// TwinCAT 3 PLC project SPT_Base_Types
// Title: SPT Base Types
// Company: Beckhoff Automation LLC
// ProjectVersion: 4.0.0.2
// Description: 4.0.0.2 I_InterfaceBase Generic base created 4.0.0.1 - removing other libs code
// libraries:
//   SPT Event Logger, * (Beckhoff Automation LLC)
//   Tc2_EtherCAT, * (Beckhoff Automation GmbH)
//   Tc2_Standard, * (Beckhoff Automation GmbH)
//   Tc2_System, * (Beckhoff Automation GmbH)
//   Tc2_Utilities, * (Beckhoff Automation GmbH)
//   Tc3_EventLogger, * (Beckhoff Automation GmbH)
//   Tc3_JsonXml, * (Beckhoff Automation GmbH)
//   Tc3_PackML_V2, * (Beckhoff Automation GmbH)
// project tree:
//   Enums/ E_AlarmResponse.TcTLEO
//   Framework Base/ FB_BaseFB.TcPOU, FB_CyclicFB.TcPOU
//   / GlobalTextList.TcGTLO, Parameters_Tracing.TcGVL
//   Interfaces/ I_BaseFB.TcIO, I_CyclicFB.TcIO, I_InterfaceBase.TcIO
//   Project Information/ F_GetCompany.TcPOU, F_GetTitle.TcPOU, F_GetVersion.TcPOU
//   Tracing/ FB_TraceLog.TcPOU, Tracing.TcGVL
//   Version/ Global_Version.TcGVL
// real-time tasks:
//   TASK Task 3: cycle T#10ms, priority 1, ADS port 350

// ---- Enums/E_AlarmResponse.TcTLEO
{attribute 'qualified_only'}
{attribute 'strict'}
{attribute 'to_string'}
TYPE E_AlarmResponse : (
		Abort_ImmediateError,
		Abort_Immediate,
		Stop_Immediate,
		Stop_Controlled,
		Hold_Immediate,
		Hold_Controlled,
		Suspend_Immediate,
		Suspend_Controlled,
		NoResponse
	);
END_TYPE

// ---- Parameters_Tracing.TcGVL
{attribute 'qualified_only'}
VAR_GLOBAL CONSTANT
	TRACING_ENABLED						: BOOL	:= TRUE;
	MAX_LOG_ENTRIES_PER_SCAN			: UDINT := 100;
	ALLOW_DUPLICATE_SEQUENTIAL_MESSAGES : BOOL	:= FALSE;
END_VAR

// ---- Tracing/Tracing.TcGVL
{attribute 'qualified_only'}
VAR_GLOBAL
	GlobalTraceLog : FB_TraceLog;
END_VAR

// ---- Version/Global_Version.TcGVL
{attribute 'TcGenerated'}
{attribute 'no-analysis'}
{attribute 'linkalways'}
// This function has been automatically generated from the project information.
VAR_GLOBAL CONSTANT
	{attribute 'const_non_replaced'}
	stLibVersion_SPT_Base_Types : ST_LibVersion := (iMajor := 4, iMinor := 0, iBuild := 0, iRevision := 2, nFlags := 0, sVersion := '4.0.0.2');
END_VAR

// ---- Interfaces/I_BaseFB.TcIO
INTERFACE I_BaseFB EXTENDS I_InterfaceBase

PROPERTY Busy : BOOL
GET
END_GET
END_PROPERTY

PROPERTY Error : BOOL
GET
END_GET
END_PROPERTY

PROPERTY ErrorID : UDINT;
GET
END_GET
END_PROPERTY

END_INTERFACE

// ---- Interfaces/I_CyclicFB.TcIO
INTERFACE I_CyclicFB EXTENDS I_BaseFB

METHOD CyclicLogic
VAR_INPUT
END_VAR
END_METHOD

PROPERTY InitComplete : BOOL
GET
END_GET
END_PROPERTY

END_INTERFACE

// ---- Interfaces/I_InterfaceBase.TcIO
INTERFACE I_InterfaceBase EXTENDS __SYSTEM.IQueryInterface

END_INTERFACE

// ---- Tracing/FB_TraceLog.TcPOU
FUNCTION_BLOCK FINAL FB_TraceLog
VAR
  Event : FB_TcMessage;
  JsonParser : FB_JsonDomParser;
  TimeFormatter : FB_FormatString;
  MessagesSentThisScan : UDINT;
  Previous_AddEntrySource : T_MaxString;
  Previous_AddEntryMessage : T_MaxString;
  Previous_AddEntryFlags : UDINT;
  Previous_AddEntryJsonSource : T_MaxString;
  Previous_AddEntryJsonMessage : T_MaxString;
  Previous_AddEntryJsonFlags : UDINT;
  Previous_AddEntryJson : T_MaxString;
END_VAR

METHOD PRIVATE AddContext
VAR_INPUT
  Source : T_MaxString;
  Flags : UDINT;
END_VAR

VAR
  CurrentDCTime : DCTIMESTRUCT;
  DCTime100Nsec : WORD;
END_VAR
//Collect DC timestamp info and properly format string
CurrentDCTime := DCTIME64_TO_DCTIMESTRUCT(F_GetActualDcTime64());
DCTime100Nsec := CurrentDCTime.wNanoseconds / 100;
TimeFormatter(
  sFormat := '%2.2d:%2.2d:%2.2d.%3.3d%3.3d%1.1d',
  arg1 := F_WORD(CurrentDCTime.wHour),
  arg2 := F_WORD(CurrentDCTime.wMinute),
  arg3 := F_WORD(CurrentDCTime.wSecond),
  arg4 := F_WORD(CurrentDCTime.wMilliseconds),
  arg5 := F_WORD(CurrentDCTime.wMicroseconds),
  arg6 := F_WORD(DCTime100Nsec)
);

Event.ipArguments.AddString(TimeFormatter.sOut); //DC Timestamp string
Event.ipArguments.AddString(Source); //POU calling the Trace() function -- this should come automatically
Event.ipArguments.AddString(TwinCAT_SystemInfoVarList._TaskInfo[GETCURTASKINDEXEX()].TaskName); //Task which called the POU last
Event.ipArguments.AddUDInt(TwinCAT_SystemInfoVarList._TaskInfo[GETCURTASKINDEXEX()].CycleCount); //Cycle count of above task
Event.ipArguments.AddUDInt(Flags); //General-use flags (application dependent)
END_METHOD

METHOD PUBLIC AddEntry
VAR_INPUT
  Source : T_MaxString;
  Message : T_MaxString;
  Flags : UDINT;
END_VAR
{analysis -62}
IF NOT TracingAllowed THEN
  {analysis -90}
  RETURN;
END_IF

IF NOT Parameters_Tracing.ALLOW_DUPLICATE_SEQUENTIAL_MESSAGES THEN
  IF (MEMCMP(ADR(Source), ADR(Previous_AddEntrySource), SIZEOF(T_MaxString)) = 0)
       AND (MEMCMP(ADR(Message), ADR(Previous_AddEntryMessage), SIZEOF(T_MaxString)) = 0)
       AND (Flags = Previous_AddEntryFlags) THEN
    //This message is identical to the last message sent--ignore
    RETURN;
  END_IF
END_IF

Event.ipArguments.Clear().AddString(Message);
AddContext(Source := Source, Flags := Flags);
Event.Send(0);
MessagesSentThisScan := MessagesSentThisScan + 1;
MEMCPY(ADR(Previous_AddEntrySource), ADR(Source), SIZEOF(T_MaxString));
MEMCPY(ADR(Previous_AddEntryMessage), ADR(Message), SIZEOF(T_MaxString));
Previous_AddEntryFlags := Flags;
END_METHOD

METHOD PUBLIC AddEntryWithJson
VAR_INPUT
  Source : T_MaxString;
  Message : T_MaxString;
  Flags : UDINT;
  Json : T_MaxString;
END_VAR

VAR
  Document : SJsonValue;
  JsonAttribute : T_MaxString;
  TaskName : T_MaxString;
  temp : udint;
END_VAR

VAR_INST
  LastScanCount : UDINT;
  MessagesSentThisScan : UDINT;
  MissedMessages : UDINT;
  Throttled : BOOL;
END_VAR

VAR
  ThrottledNotificationString : T_MaxString;
  CurrentDCTime : DCTIMESTRUCT;
  DCTime100Nsec : WORD;
  DCTimeString : T_MaxString;
END_VAR
{analysis -62}
IF NOT TracingAllowed THEN
  RETURN;
END_IF

IF NOT Parameters_Tracing.ALLOW_DUPLICATE_SEQUENTIAL_MESSAGES THEN
  IF (MEMCMP(ADR(Source), ADR(Previous_AddEntryJsonSource), SIZEOF(T_MaxString)) = 0)
       AND (MEMCMP(ADR(Message), ADR(Previous_AddEntryJsonMessage), SIZEOF(T_MaxString)) = 0)
       AND (Flags = Previous_AddEntryJsonFlags)
       AND (MEMCMP(ADR(Json), ADR(Previous_AddEntryJson), SIZEOF(T_MaxString)) = 0) THEN
    //This message is identical to the last message sent--ignore
    RETURN;
  END_IF
END_IF

Event.ipArguments.Clear().AddString(Message);
AddContext(Source := Source, Flags := Flags);
Document := JsonParser.NewDocument();
JsonParser.AddJsonMember(Document, 'ExtendedInfo', Json);
JsonAttribute := JsonParser.GetJson(Document);
Event.SetJsonAttribute(JsonAttribute);
Event.Send(0);
MessagesSentThisScan := MessagesSentThisScan + 1;
MEMCPY(ADR(Previous_AddEntryJsonSource), ADR(Source), SIZEOF(T_MaxString));
MEMCPY(ADR(Previous_AddEntryJsonMessage), ADR(Message), SIZEOF(T_MaxString));
Previous_AddEntryFlags := Flags;
MEMCPY(ADR(Previous_AddEntryJsonMessage), ADR(Json), SIZEOF(T_MaxString));
END_METHOD

METHOD FB_init : BOOL
VAR_INPUT
  bInitRetains : BOOL; // if TRUE, the retain variables are initialized (warm start / cold start)
  bInCopyCode : BOOL; // if TRUE, the instance afterwards gets moved into the copy code (online change)
END_VAR

VAR
  hr : HRESULT;
END_VAR
{analysis -15}
IF NOT Event.EqualsToEventEntryEx(TC_EVENTS.Tracing.TraceEvent) THEN
  Event.CreateEx(TC_EVENTS.Tracing.TraceEvent, 0);
END_IF
END_METHOD

PROPERTY PRIVATE TracingAllowed : BOOL
GET
VAR_INST
  LastScanCount : UDINT;
  MissedMessages : UDINT;
  Throttled : BOOL;
END_VAR

VAR
  ThrottledNotificationString : T_MaxString;
END_VAR
{analysis -62}
IF NOT Parameters_Tracing.TRACING_ENABLED THEN
  TracingAllowed := FALSE;
  RETURN;
END_IF

IF TwinCAT_SystemInfoVarList._TaskInfo[GETCURTASKINDEXEX()].CycleCount = LastScanCount THEN
  //Trying to send multiple messages in same scan
  IF Throttled THEN
    MissedMessages := MissedMessages + 1;
    RETURN;
  ELSIF MessagesSentThisScan >= Parameters_Tracing.MAX_LOG_ENTRIES_PER_SCAN AND NOT Throttled THEN
    //Need to throttle messsage queue
    Event.ipArguments.Clear().AddString('Too many messages sent in single scan; tracing throttled.');
    Event.Send(0);
    MissedMessages := MissedMessages + 1;
    Throttled := TRUE;
    TracingAllowed := FALSE;
    RETURN;
  ELSE
    TracingAllowed := TRUE;
  END_IF
ELSE
  IF Throttled THEN
    ThrottledNotificationString := CONCAT('Missed ', CONCAT(TO_STRING(MissedMessages), ' throttled messages previously.'));
    Event.ipArguments.Clear().AddString(ThrottledNotificationString);
    Event.Send(0);
    MissedMessages := 0;
  END_IF

  LastScanCount := TwinCAT_SystemInfoVarList._TaskInfo[GETCURTASKINDEXEX()].CycleCount;
  MessagesSentThisScan := 0;
  Throttled := FALSE;
  TracingAllowed := TRUE;
END_IF
END_GET
END_PROPERTY

END_FUNCTION_BLOCK

// ---- Framework Base/FB_BaseFB.TcPOU
{attribute 'reflection'}
FUNCTION_BLOCK ABSTRACT FB_BaseFB IMPLEMENTS I_BaseFB
VAR
  {attribute 'instance-path'}
  {attribute 'noinit'}
  InstancePath : STRING;
END_VAR

// I_BaseFB
VAR
  _Busy : BOOL := TRUE;
  _Error : BOOL;
  _ErrorID : UDINT;
END_VAR

// Derivatives of FB_BaseFB can have code in the function block body

PROPERTY Busy : BOOL
GET
Busy := _Busy;
END_GET
END_PROPERTY

PROPERTY Error : BOOL
GET
Error := _Error;
END_GET
END_PROPERTY

PROPERTY ErrorID : UDINT
GET
ErrorID := _ErrorID;
END_GET
END_PROPERTY

METHOD PUBLIC Marker
VAR_INPUT
  Message : T_MaxString;
END_VAR
Tracing.GlobalTraceLog.AddEntry(InstancePath, Message, 1);
END_METHOD

METHOD PUBLIC Trace
VAR_INPUT
  Message : T_MaxString;
END_VAR
Tracing.GlobalTraceLog.AddEntry(InstancePath, Message, 0);
END_METHOD

METHOD PUBLIC TraceWithJson
VAR_INPUT
  Message : T_MaxString;
  Json : T_MaxString;
END_VAR
Tracing.GlobalTraceLog.AddEntryWithJson(
  InstancePath,
  Message,
  0,
  Json
);
END_METHOD

END_FUNCTION_BLOCK

// ---- Framework Base/FB_CyclicFB.TcPOU
{attribute 'no_call'}
FUNCTION_BLOCK ABSTRACT FB_CyclicFB EXTENDS FB_BaseFB IMPLEMENTS I_CyclicFB
VAR
  _InitComplete : BOOL;
END_VAR

// Derivatives of FB_CyclicFB should *NOT* have code in the function block body

// Use CyclicLogic() instead

METHOD PUBLIC ABSTRACT CyclicLogic
VAR_INPUT
END_VAR
END_METHOD

PROPERTY InitComplete : BOOL
GET
InitComplete := _InitComplete;
END_GET
END_PROPERTY

END_FUNCTION_BLOCK

// ---- Project Information/F_GetCompany.TcPOU
// This function has been automatically generated from the project information.
{attribute 'signature_flag' := '1073741824'}
{attribute 'TcGenerated'}
{attribute 'no-analysis'}
FUNCTION F_GetCompany : WSTRING
VAR_INPUT
	
END_VAR

F_GetCompany := "Beckhoff Automation LLC";

END_FUNCTION

// ---- Project Information/F_GetTitle.TcPOU
// This function has been automatically generated from the project information.
{attribute 'signature_flag' := '1073741824'}
{attribute 'TcGenerated'}
{attribute 'no-analysis'}
FUNCTION F_GetTitle : WSTRING
VAR_INPUT
	
END_VAR

F_GetTitle := "SPT Base Types";

END_FUNCTION

// ---- Project Information/F_GetVersion.TcPOU
// This function has been automatically generated from the project information.
{attribute 'signature_flag' := '1073741824'}
{attribute 'TcGenerated'}
{attribute 'no-analysis'}
FUNCTION F_GetVersion : ST_LibVersion
VAR_INPUT
	
END_VAR

F_GetVersion.iMajor := 4;
F_GetVersion.iMinor := 0;
F_GetVersion.iBuild := 0;
F_GetVersion.iRevision := 2;
F_GetVersion.sVersion := '4.0.0.2';
F_GetVersion.nFlags := 0;

END_FUNCTION

// ---- GlobalTextList.TcGTLO
TEXTLIST GlobalTextList
  685 = '%s'
  680 = 'Abort'
  452 = 'Clear'
  744 = 'Hold'
  347 = 'MACHINE'
  46 = 'Maintenance'
  904 = 'Manual'
  929 = 'Production'
  181 = 'Reset'
  77 = 'Start'
  516 = 'State: %s'
  828 = 'Stop'
  806 = 'Suspend'
  197 = 'Unhold'
  832 = 'Unsuspend'
END_TEXTLIST
